ABB RobotStudio station: ABB_Pick_and_place_sol_1.rspag

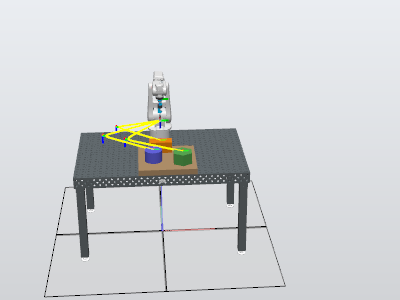
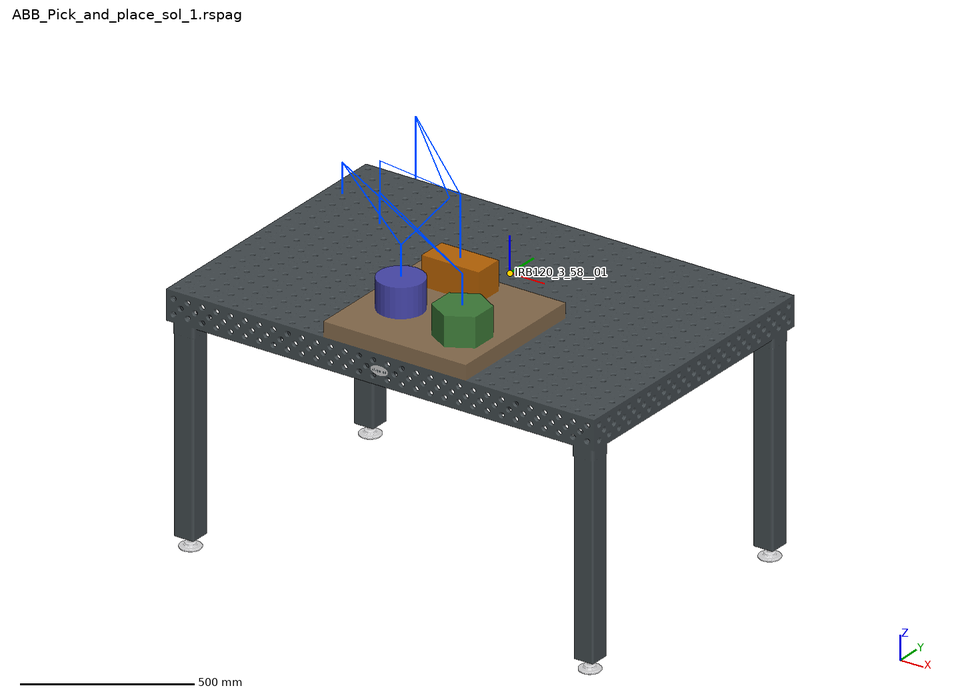
[picture v1: parts stored in the station drawn from their meshes, with robot base, taught points and paths (robot models come from the ABB library and are not in the file)]
--- station ---
Station FINAL FUCKING TRY (saved by RobotStudio 22.3.10190.2)
Controller Controller1, task T_ROB1: task frame (RAPID world) sits at (0, 150, 830) mm, rotated rx 0 ry 0 rz -90 deg in the station
Controller Controller1
  mechanical unit ROB_1: IRB120_3_58__01, 6 joints, base frame (0, 0, 0) mm
Layout (positions relative to the parent item):
  - table [part] at (-200, -500, 830) mm, size 500 x 500 x 50 mm
  - object_1 [part] at (-200, -500, 830) mm, size 200 x 100 x 150 mm
  - object_2 [part] at (-200, -500, 830) mm, size 149.5 x 149.7 x 150 mm
  - object_3 [part] at (-200, -500, 830) mm, size 155.5 x 179.5 x 150 mm
  - siegmund_1500_1000 [part], size 1500 x 1010.3 x 830 mm
  - object_11 [part] at (-200, -500, 830) mm, size 200 x 100 x 150 mm
  - object_22 [part] at (-200, -500, 830) mm, size 149.5 x 149.7 x 150 mm
  - object_33 [part] at (-200, -500, 830) mm, size 155.5 x 179.5 x 150 mm
  - IRB120_3_58__01 [mechanism, from Robots\IRB120_3_58_G_01.rslib] at (0, 150, 830) mm, rotated rx 0 ry 0 rz -90 deg; joint values [0, 0, 0, 0, 1.5708, 0] (rad or m)
  - smc_gripper [mechanism, from Gripper_RS_tool\smc_gripper.rslib] at (0, -152, 1388) mm, rotated rx 180 ry 0 rz 90 deg
  - Positioner [smart component, from Components\Positioner.rslib]
      properties: Object=object_1; Position=[-0.6 -0.15 0.83]; Orientation=[0 0 0]; Reference=Global; ReferenceObject=(none)
  - Positioner_2 [smart component, from Components\Positioner.rslib]
      properties: Object=object_2; Position=[-0.65 -0.15 0.83]; Orientation=[0 0 0]; Reference=Global; ReferenceObject=(none)
  - Positioner_3 [smart component, from Components\Positioner.rslib]
      properties: Object=object_3; Position=[-0.7 -0.2 0.83]; Orientation=[0 0 0]; Reference=Global; ReferenceObject=(none)
  - Attacher [smart component, from Components\Attacher.rslib]
      properties: Parent=smc_gripper; Flange=0; Child=object_1; Mount=false; Offset=[0 0 0]; Orientation=[0 0 0]
  - Attacher_2 [smart component, from Components\Attacher.rslib]
      properties: Parent=smc_gripper; Flange=0; Child=object_2; Mount=false; Offset=[0 0 0]; Orientation=[0 0 0]
  - Attacher_3 [smart component, from Components\Attacher.rslib]
      properties: Parent=smc_gripper; Flange=0; Child=object_3; Mount=false; Offset=[0 0 0]; Orientation=[0 0 0]
  - Detacher [smart component, from Components\Detacher.rslib]
      properties: Child=object_1; KeepPosition=true
  - Detacher_2 [smart component, from Components\Detacher.rslib]
      properties: Child=object_2; KeepPosition=true
  - Detacher_3 [smart component, from Components\Detacher.rslib]
      properties: Child=object_3; KeepPosition=true
Attachment: smc_gripper is attached to IRB120_3_58__01 / Link6
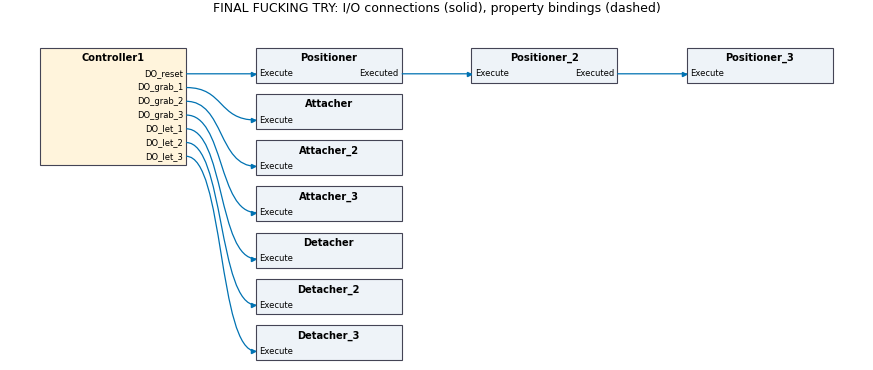
Station logic (signal -> signal, property => property):
  Controller1.DO_reset -> Positioner.Execute
  Positioner.Executed -> Positioner_2.Execute
  Positioner_2.Executed -> Positioner_3.Execute
  Controller1.DO_grab_1 -> Attacher.Execute
  Controller1.DO_grab_2 -> Attacher_2.Execute
  Controller1.DO_grab_3 -> Attacher_3.Execute
  Controller1.DO_let_1 -> Detacher.Execute
  Controller1.DO_let_2 -> Detacher_2.Execute
  Controller1.DO_let_3 -> Detacher_3.Execute
Targets, tools, work objects and paths stored in the station and not in the controller backup, written as RAPID:
! task T_ROB1
MODULE Module1
  PROC Path_10()
    MoveL home,v1000,z100,smc_gripper\WObj:=wobj0;
    MoveL o_home,v1000,z100,smc_gripper\WObj:=wobj0;
    MoveL o_goal,v1000,z100,smc_gripper\WObj:=wobj0;
  ENDPROC
  PROC Path_20()
    MoveL home,v1000,z100,smc_gripper\WObj:=wobj0;
    MoveL b_home,v1000,z100,smc_gripper\WObj:=wobj0;
    MoveL b_goal,v1000,z100,smc_gripper\WObj:=wobj0;
  ENDPROC
  PROC Path_30()
    MoveL home,v1000,z100,smc_gripper\WObj:=wobj0;
    MoveL g_home,v1000,z100,smc_gripper\WObj:=wobj0;
    MoveL g_goal,v1000,z100,smc_gripper\WObj:=wobj0;
  ENDPROC
ENDMODULE


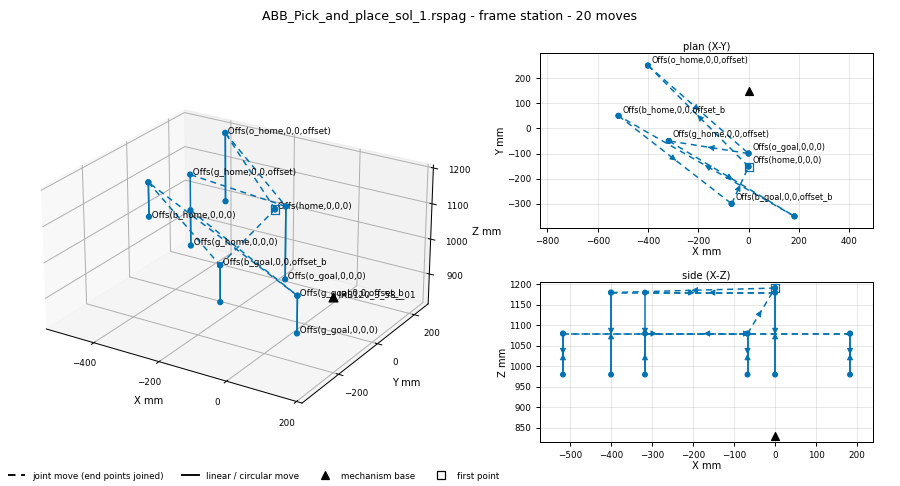
[picture p0: tool path of ABB_Pick_and_place_sol_1.rspag in frame station, 20 of 20 moves have a stored position in this frame; points joined in program order, loops and branches not executed]
--- Backups/Controller1/RAPID/TASK1/PROGMOD/CalibData.mod ---
MODULE CalibData
    PERS tooldata smc_gripper:=[TRUE,[[0,0.004,197.001],[1,0,0,0]],[1,[0.207,-0.496,71.18],[1,0,0,0],0,0,0]];
ENDMODULE

--- Backups/Controller1/RAPID/TASK1/PROGMOD/Module1.mod ---
MODULE Module1
        CONST robtarget home:=[[302,0.004,360.999],[0,0,1,0],[-1,0,-1,0],[9E+09,9E+09,9E+09,9E+09,9E+09,9E+09]];
    CONST robtarget o_home:=[[-100,-400,150],[0,0,1,0],[0,0,0,0],[9E+09,9E+09,9E+09,9E+09,9E+09,9E+09]];
    CONST robtarget o_goal:=[[250,0,150],[0,0,1,0],[0,0,0,0],[9E+09,9E+09,9E+09,9E+09,9E+09,9E+09]];
    CONST robtarget b_home:=[[100,-517.298,150],[0,0,1,0],[0,0,0,0],[9E+09,9E+09,9E+09,9E+09,9E+09,9E+09]];
    CONST robtarget b_goal:=[[450,-67.298,150],[0,0,1,0],[0,0,0,0],[9E+09,9E+09,9E+09,9E+09,9E+09,9E+09]];
    CONST robtarget g_home:=[[200,-317.298,150],[0,0,1,0],[0,0,0,0],[9E+09,9E+09,9E+09,9E+09,9E+09,9E+09]];
    CONST robtarget g_goal:=[[500,182.702,150],[0,0,1,0],[0,0,0,0],[9E+09,9E+09,9E+09,9E+09,9E+09,9E+09]];
    VAR num offset := 200;
    VAR num offset_b := 100;

    PROC main()
        !prep
        PulseDO DO_let_1;
        PulseDO DO_let_2;
        PulseDO DO_let_3;
        PulseDO DO_reset;
        MoveJ Offs(home,0,0,0),v1000,fine,smc_gripper;

        !orange
        MoveJ Offs(o_home,0,0,offset),v1000,z100,smc_gripper;
        MoveL Offs(o_home,0,0,0),v100,fine,smc_gripper;
        WaitTime 1.0;
        PulseDO DO_grab_1;
        MoveL Offs(o_home,0,0,offset),v100,fine,smc_gripper;
        MoveJ Offs(o_goal,0,0,offset),v1000,z100,smc_gripper;
        MoveL Offs(o_goal,0,0,0),v100,fine,smc_gripper;
        WaitTime 1.0;
        PulseDO DO_let_1;
        MoveL Offs(o_goal,0,0,offset),v100,fine,smc_gripper;

        !green
        MoveJ Offs(g_home,0,0,offset),v1000,z100,smc_gripper;
        MoveL Offs(g_home,0,0,0),v100,fine,smc_gripper;
        WaitTime 1.0;
        PulseDO DO_grab_3;
        MoveL Offs(g_home,0,0,offset_b),v100,fine,smc_gripper;
        MoveJ Offs(g_goal,0,0,offset_b),v1000,z100,smc_gripper;
        MoveL Offs(g_goal,0,0,0),v100,fine,smc_gripper;
        WaitTime 1.0;
        PulseDO DO_let_3;
        MoveL Offs(g_goal,0,0,offset_b),v100,fine,smc_gripper;

        !blue
        MoveJ Offs(b_home,0,0,offset_b),v1000,z100,smc_gripper;
        MoveL Offs(b_home,0,0,0),v100,fine,smc_gripper;
        WaitTime 1.0;
        PulseDO DO_grab_2;
        MoveL Offs(b_home,0,0,offset_b),v100,fine,smc_gripper;
        MoveJ Offs(b_goal,0,0,offset_b),v1000,z100,smc_gripper;
        MoveL Offs(b_goal,0,0,0),v100,fine,smc_gripper;
        WaitTime 1.0;
        PulseDO DO_let_2;
        MoveL Offs(b_goal,0,0,offset_b),v100,fine,smc_gripper;

        MoveJ Offs(home,0,0,0),v1000,fine,smc_gripper;

    ENDPROC

ENDMODULE

--- Backups/Controller1/SYSPAR/EIO.cfg ---
EIO:CFG_1.0:6:1::
#
EIO_SIGNAL:

      -Name "DO_reset" -SignalType "DO"

      -Name "DO_grab_1" -SignalType "DO"

      -Name "DO_grab_2" -SignalType "DO"

      -Name "DO_grab_3" -SignalType "DO"

      -Name "DO_let_1" -SignalType "DO"

      -Name "DO_let_2" -SignalType "DO"

      -Name "DO_let_3" -SignalType "DO"
